(* IEC 61131-3 sources: go-native-ads/examples/rpc/plc, 3 files *)

(* ---- FB_RPC.st ---- *)
FUNCTION_BLOCK FB_RPC
VAR
    calls : UDINT;
END_VAR

(* ---- Add.st ---- *)
{attribute 'TcRpcEnable'}
METHOD PUBLIC Add : INT
VAR_INPUT
    a : INT;
    b : INT;
END_VAR

Add := a + b;
calls := calls + 1;

(* ---- MAIN.st ---- *)
PROGRAM MAIN
VAR
    rpc : FB_RPC;
END_VAR

rpc();
